(* IEC 61131-3 sources: Summary-ETFA22/ahorn/benchmark/PLCopen/library, 3 files *)

(* ---- F_TRIG.st ---- *)
FUNCTION_BLOCK F_TRIG
VAR_INPUT
   CLK: BOOL;
END_VAR
VAR_OUTPUT
   Q: BOOL;
END_VAR
VAR
   M: BOOL;
END_VAR
Q := NOT CLK AND M;
M := CLK;
END_FUNCTION_BLOCK

(* ---- R_TRIG.st ---- *)
FUNCTION_BLOCK R_TRIG
VAR_INPUT
   CLK: BOOL;
END_VAR
VAR_OUTPUT
   Q: BOOL;
END_VAR
VAR
   M: BOOL;
END_VAR
Q := CLK AND NOT M;
M := CLK;
END_FUNCTION_BLOCK

(* ---- TON.st ---- *)
FUNCTION_BLOCK TON
VAR_INPUT
    IN : BOOL;
    PT : TIME;
END_VAR
VAR_OUTPUT
      Q : BOOL;
END_VAR
IF NOT IN THEN
    Q := FALSE;
ELSIF NOT Q THEN
    Q := NONDETERMINISTIC_BOOL();
END_IF;
END_FUNCTION_BLOCK
